// TIA Portal V18 export
TYPE "udtVciBG"
// stored: IsFailsafeCompliant false
   STRUCT
      setTimeTon : Time;
      setTimeTof : Time;
      GetTimeTonElapsed : Time;
      GetTimeTofElapsed : Time;
      GetActualState : Bool;
   END_STRUCT;
END_TYPE
